TYPE DUT :
UNION
	

bit1	: BOOL;
bit2	: BOOL;
bit3	: BOOL;
bit4	: BOOL;

byte1	: BYTE;



END_UNION
END_TYPE

(* stored: Version 1.1.0.1, ProductVersion 3.1.4024.12
   DUT DUT: Id {1461dfae-5b45-4976-8e93-4d3d5ba93aae} *)
